// Annex I I.10 - the help points serving one nest. Count = 1 is the trivial
// single-help case; multi-help is the general one.
TYPE ST_NestHelpAffinity :
STRUCT
    Helps : ARRAY[1..PL_RobotPlanner.MAX_HELPS_PER_NEST] OF ST_HelpAffinity;
    Count : INT;
END_STRUCT
END_TYPE

(* stored: Version 1.1.0.1, ProductVersion 3.1.4024.12
   DUT ST_NestHelpAffinity: Id {e37b52ed-66b6-4229-8604-f84f0399e4c1} *)
